Fanuc KAREL source: ko00084.KL

-- PROVISIONAL review KL for V940-1; original PC SHA256 bac0b0716ce9a322269079ae6586890a54dc52dacc5e9ad8a0eea8f4ed6fb42f
-- Incomplete behavior may be omitted. Consult companion uncertainty JSON. Do not deploy.
PROGRAM KO00084
%NOLOCKGROUP
BEGIN
  -- V9_ZERO_TABLE_METADATA_HINT layout=0002_ascii; no indexed target words; source/name/runtime held
  -- UNRESOLVED_PC offsets 5-12; opcodes 9D,23
  -- UNRESOLVED_PC offsets 17-66; opcodes 27,27,49,7E,AD,22,1C,22,31,7E,4A
  -- UNRESOLVED_PC offsets 71-75; opcodes 7F
END KO00084
